PROGRAM TextDisplay
VAR
	TextDis: STRING;
END_VAR

IF GVL.ixSensor1 THEN
	TextDis := 'Home';
ELSIF
	GVL.ixSensor2 THEN
	TextDis := 'Station 1';
ELSIF GVL.qxButtEmerg AND NOT GVL.qxButtRight AND NOT GVL.qxButtLeft THEN
	TextDis := 'Emergency Stop';
ELSE
	TextDis := 'Moving';
END_IF

END_PROGRAM

(* stored: Version 1.1.0.1, ProductVersion 3.1.4024.12
   POU TextDisplay: Id {085e54ff-aae8-4497-9340-166d4a684833}, SpecialFunc None *)
